{attribute addProperty BoxType "EL3051-0000-0016"}
{attribute addProperty Id "AI_StandardAT %I*AI_Standard_BC62E3BB7290WcStateAT %I*WcState_F855686C1620InfoDataAT %I*InfoData_BC63D37F80100"}
{attribute addProperty CRC "2549024560"}
{attribute addProperty SizeInBites "168"}
{attribute addProperty SizeInBytes "21"}
TYPE EL3051_EE4FF550 :
STRUCT
	{attribute addProperty Name "AI_Standard"}
	AI_Standard : AI_Standard_BC62E3BB;
	{attribute addProperty Name "WcState"}
	WcState : WcState_F855686C;
	{attribute addProperty Name "InfoData"}
	InfoData : InfoData_BC63D37F;
END_STRUCT
END_TYPE

(* stored: Version 1.2.0.0, ProductVersion 3.1.4024.9
   DUT EL3051_EE4FF550: Id {5a4bc96f-c3ef-4c46-bdfe-22129e5b25be} *)
